FUNCTION_BLOCK StringBufferOutput IMPLEMENTS IStringBufferOutput
VAR_INPUT
END_VAR
VAR_OUTPUT
END_VAR
VAR
  output_message: STRING(255);
END_VAR

METHOD compose_message
VAR_INPUT
  message: STRING(80);
END_VAR
output_message := CONCAT(output_message, message);
END_METHOD

METHOD get_output : STRING(255)
get_output := output_message;
END_METHOD

END_FUNCTION_BLOCK

(* stored: Version 1.1.0.1, ProductVersion 3.1.4022.7
   POU StringBufferOutput: Id {96897f13-93b5-4bf7-8010-d68bee21eb01}, SpecialFunc None
   Method compose_message: Id {ca98fe10-be10-412e-96f4-82fb32511f65}
   Method get_output: Id {e7610127-b8e7-41df-b955-7e3d2ba2a002} *)
